% RSLogix 500 project REJECT_TRACKING_B.RSS, saved by version 8.30.00.16 %
PROJECT "UNTITLED"    % processor: Bul.1763 MicroLogix 1100 Series B %

PROGRAM FILES
  LAD 2   6 rungs

DATA FILES
  O0 OUTPUT  4 elements
  I1 INPUT  6 elements
  S2 STATUS  66 elements
  B3 BINARY  10 elements
  T4 TIMER  5 elements
  C5 COUNTER  5 elements
  R6 CONTROL  1 elements
  N7 INTEGER  1 elements
  F8 FLOAT  1 elements
  B93 BIT_ARRAY  4 elements  % Binary Bit Array %
  N199 NUM_BOXES  5 elements  % Number of Boxes in Between PE1 & PE2 %

LADDER 2
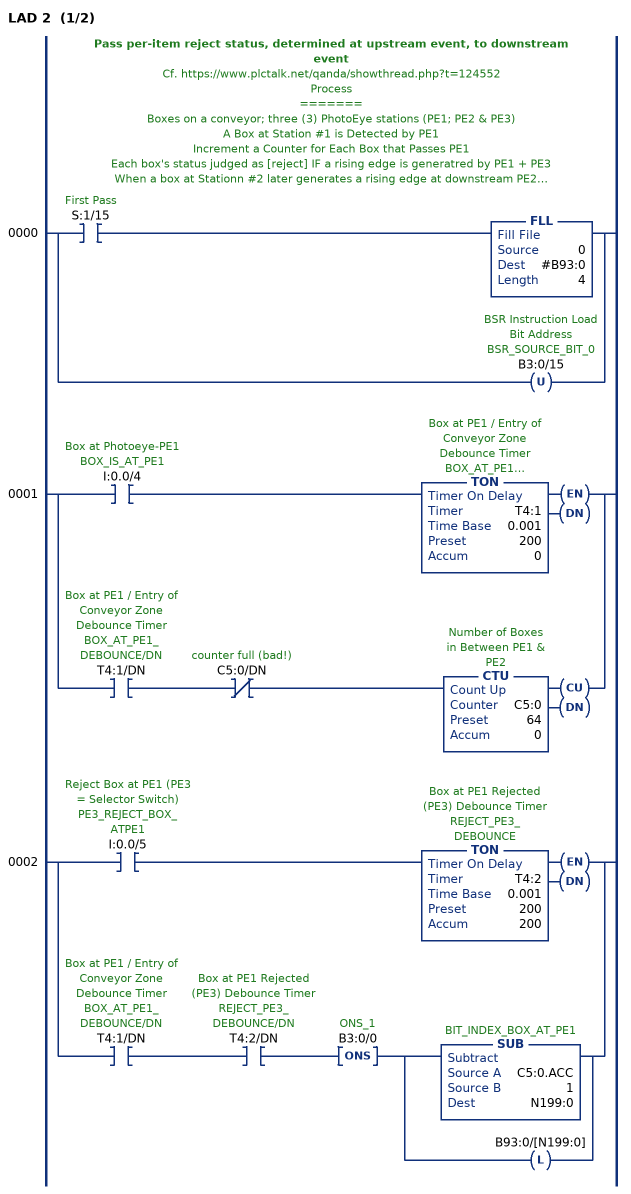
% Rung: 0 %
% TITLE: Pass per-item reject status, determined at upstream event, to downstream event %
% Cf. https://www.plctalk.net/qanda/showthread.php?t=124552
% 
% Process
% =======
% Boxes on a conveyor; three (3) PhotoEye stations (PE1; PE2 & PE3)
% A Box at Station #1 is Detected by PE1
% Increment a Counter for Each Box that Passes PE1
% Each box's status judged as [reject] IF a rising edge is generatred by PE1 + PE3
% When a box at Stationn #2 later generates a rising edge at downstream PE2:
% - divert if box status from PE1 + PE3 was [reject]
% - do not divert if box status from PE1 was [okay]
% Decrement a Counter for Each Box that is detected by at Station #2 (PE2)
% 
% Implementation summary
% ====================
% Pulse BSR with PE2 to Shift the Bit Array
% BSR Length = number of boxes from PE1 to before PE2
% 
% N.B. Assumptions
% - Adequate space between boxes, so 1 rising edge per box at PE1 and at PE2
% - No boxed added or subtracted between PE1 and PE2 (or coffee cup blocks PE)
% - PE1 & PE3 are positioned so a Box Enterng the Station #1 to Station#2 Zone (PE1) & a Rejected Box (PE3) can detect each condition at the same time
% 
% Initialization
% =========
% - Set FIFO Bit Array and index pointers to zero
% - Unlatch the BSR Load Bit (B3:0/15) because it is must be 0 when pushed onto the top of the FIFO Bit Array %
SOR BST XIC S:1/15 FLL 0 #B93:0 4 NXB OTU B3:0/15 BND EOR
%   S:1/15  "First Pass" %
%   B3:0/15  BSR_SOURCE_BIT_0  "BSR Instruction Load Bit Address" %
% Rung: 1 %
SOR BST XIC I:0.0/4 TON T4:1 0.001 200 0 NXB XIC T4:1/DN XIO C5:0/DN CTU C5:0 64 0 BND EOR
%   I:0.0/4  BOX_IS_AT_PE1  "Box at Photoeye-PE1" %
%   T4:1  BOX_AT_PE1_DEBOUNCE  "Box at PE1 / Entry of Conveyor Zone Debounce Timer" %
%   C5:0/DN  "counter full (bad!)" %
%   C5:0  "Number of Boxes in Between PE1 & PE2" %
% Rung: 2 %
SOR BST XIC I:0.0/5 TON T4:2 0.001 200 200 NXB XIC T4:1/DN XIC T4:2/DN ONS B3:0/0 BST SUB C5:0.ACC 1 N199:0 NXB OTL B93:0/[N199:0] BND BND EOR
%   I:0.0/5  PE3_REJECT_BOX_ATPE1  "Reject Box at PE1 (PE3 = Selector Switch)" %
%   T4:2  REJECT_PE3_DEBOUNCE  "Box at PE1 Rejected (PE3) Debounce Timer" %
%   T4:1  BOX_AT_PE1_DEBOUNCE  "Box at PE1 / Entry of Conveyor Zone Debounce Timer" %
%   B3:0/0  ONS_1 %
%   C5:0  "Number of Boxes in Between PE1 & PE2" %
%   N199:0  BIT_INDEX_BOX_AT_PE1 %

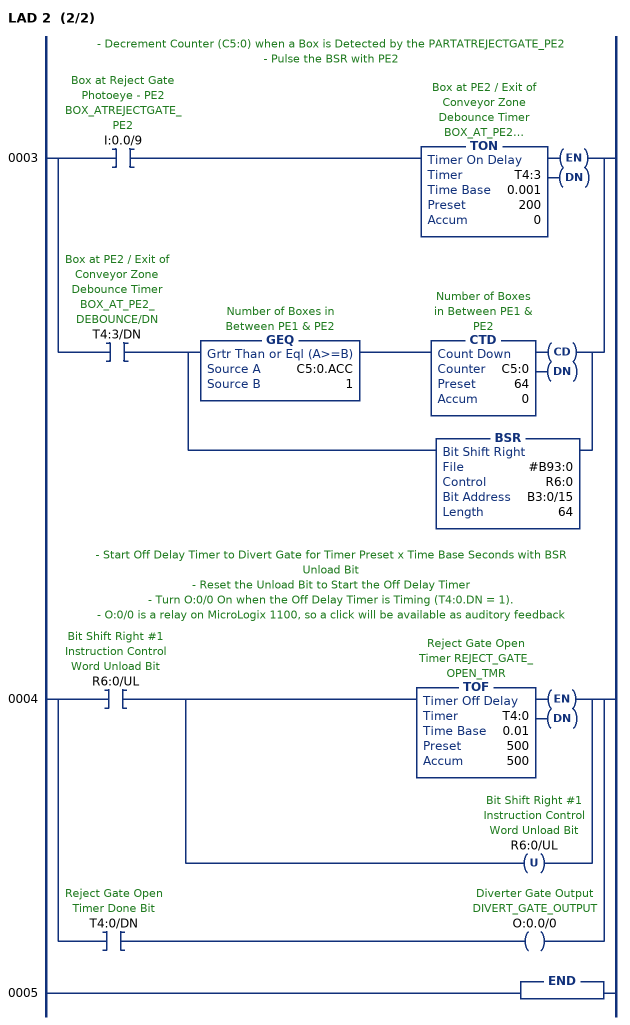
% Rung: 3 %
% - Decrement Counter (C5:0) when a Box is Detected by the PARTATREJECTGATE_PE2
% - Pulse the BSR with PE2 %
SOR BST XIC I:0.0/9 TON T4:3 0.001 200 0 NXB XIC T4:3/DN BST GEQ C5:0.ACC 1 CTD C5:0 64 0 NXB BSR #B93:0 R6:0 B3:0/15 64 BND BND EOR
%   I:0.0/9  BOX_ATREJECTGATE_PE2  "Box at Reject Gate Photoeye - PE2" %
%   T4:3  BOX_AT_PE2_DEBOUNCE  "Box at PE2 / Exit of Conveyor Zone Debounce Timer" %
%   C5:0  "Number of Boxes in Between PE1 & PE2" %
%   R6:0  BSR_1_CONTROL  "Bit Shift Right #1 Instruction Control Word" %
%   B3:0/15  BSR_SOURCE_BIT_0  "BSR Instruction Load Bit Address" %
% Rung: 4 %
% - Start Off Delay Timer to Divert Gate for Timer Preset x Time Base Seconds with BSR Unload Bit
% - Reset the Unload Bit to Start the Off Delay Timer
% - Turn O:0/0 On when the Off Delay Timer is Timing (T4:0.DN = 1).
%   - O:0/0 is a relay on MicroLogix 1100, so a click will be available as auditory feedback %
SOR BST XIC R6:0/UL BST TOF T4:0 0.01 500 500 NXB OTU R6:0/UL BND NXB XIC T4:0/DN OTE O:0.0/0 BND EOR
%   R6:0/UL  "Bit Shift Right #1 Instruction Control Word Unload Bit" %
%   T4:0  REJECT_GATE_OPEN_TMR  "Reject Gate Open Timer" %
%   T4:0/DN  "Reject Gate Open Timer Done Bit" %
%   O:0.0/0  DIVERT_GATE_OUTPUT  "Diverter Gate Output" %
% Rung: 5 %
SOR END EOR

COMMENTS NOT ATTACHED TO A CURRENT RUNG
  T4:1: Act on PE2 rising edge Part IIb
    - Changing from diverted to not-diverted
    - Unlatch diverted state
    - Start timer as proxy for sending MSG to deactivate diverter
  N199:0: Detect rising edges of PE1 / PE2 / PE3 inputs
    If PART_AT_REJECT_PE1 = 1 Then Increment the Counter (C5:0)
    IF PART_AT_REJECT_PE!1 =1 AND  REJECT_AT_PE1 (PE3 = I:0/5) Then Calculate the B93 Word Address & Bit Address & Latch That Bit On / =1 to Store the Reject Part Status at the Correct Position in the B93 Bit Array "Virtual FIFO" - Note: There are no FFL / FFU Instructions for Bit Arrays in Alleno-Bradley PLCs
    Stop Incrementing the Counter (C5:0) When the Conveyor is Full (C5:0.ACC = 63

DATA TABLE (non-zero values as saved)
DATA T4
% .PRE .ACC %
% T4:0 % 500 500
% T4:1 % 200 0
% T4:2 % 200 200
% T4:3 % 200 0
DATA C5
% .PRE .ACC %
% C5:0 % 64 0
DATA R6
% .LEN .POS %
% R6:0 % 64 0
DATA N199
% N199:0 % -1 0 0 0 0
